{attribute addProperty BoxType "KL1644-0050"}
{attribute addProperty Id "SwitchAT %I*BOOL000OutputAT %Q*BOOL000"}
{attribute addProperty CRC "2112668104"}
{attribute addProperty SizeInBites "0"}
{attribute addProperty SizeInBytes "0"}
TYPE Channel_7DECC1C8 :
STRUCT
	{attribute addProperty Name "Switch"}
	Switch AT %I* : BOOL;
	{attribute addProperty Name "Output"}
	Output AT %Q* : BOOL;
END_STRUCT
END_TYPE

(* stored: Version 1.2.0.0, ProductVersion 3.1.4024.9
   DUT Channel_7DECC1C8: Id {8e35ef4b-ee06-4067-82e8-87d633088965} *)
